FUNCTION_BLOCK FB_BalluffPosition
VAR_INPUT
END_VAR
VAR_OUTPUT
	Error	: BOOL;
	Position: REAL;
	Temperature	: REAL;
END_VAR
VAR
	Magnet AT %I* : ST_BalluffMagnet;
END_VAR

Error:= (Magnet.PosAboveWorkAreaHighLimit<>0) OR (Magnet.PosBelowWorkAreaLowLimit<>0) OR (Magnet.PosMarkerFailure<>0);
Position:= DINT_TO_REAL(Magnet.Position)/1000.0;

END_FUNCTION_BLOCK

(* stored: Version 1.1.0.1, ProductVersion 3.1.4020.12
   POU FB_BalluffPosition: Id {904ffdb5-4a0f-47a4-83f0-51f51cdb2384}, SpecialFunc None *)
